// TIA Portal V20 export
TYPE "typeFDoorUnlockOutput"
// stored: Access Published, IsFailsafeCompliant true, Namespace Safety
   STRUCT
      unwinderRearDoorUnlock : Bool;   // F Door Unlock Cmd Status
      autoSpliceDoorUnlock : Bool;   // F Door Unlock Cmd Status
      unwinderMainDoorUnlock : Bool;   // F Door Unlock Cmd Status
      unwinderTopDoorUnlock : Bool;   // F Door Unlock Cmd Status
      unwinderBtmDoorUnlock : Bool;   // F Door Unlock Cmd Status
      stackTableDoorUnlock : Bool;   // F Door Unlock Cmd Status
      jrWinderDoorOpen : Bool;   // F Door Unlock Cmd Status
   END_STRUCT;
END_TYPE
